TYPE "Positioning_EPOS_Machine_Par"
VERSION : 0.1
// Block: Positioning_EPOS_Machine_Par
   STRUCT
      PosTolerance : LReal;
      DelayInPosition : Time;
      Man_Vel : LReal;
      Man_Acc : LReal;
      Man_Dec : LReal;
   END_STRUCT;

END_TYPE
